// TIA Portal V20 export
TYPE "typeFDoorFunction"
// Safety status of door
// stored: Access Published, IsFailsafeCompliant true, Namespace Safety
   STRUCT
      fDoor1 { S7_SetPoint := 'True'} : "Safety.typeFDoorFunctionData";
      fDoor2 { S7_SetPoint := 'True'} : "Safety.typeFDoorFunctionData";   // Safety status of door
      fDoor3 { S7_SetPoint := 'True'} : "Safety.typeFDoorFunctionData";   // Safety status of door
      fDoor4 { S7_SetPoint := 'True'} : "Safety.typeFDoorFunctionData";   // Safety status of door
      fDoor5 { S7_SetPoint := 'True'} : "Safety.typeFDoorFunctionData";   // Safety status of door
      fDoor6 { S7_SetPoint := 'True'} : "Safety.typeFDoorFunctionData";   // Safety status of door
      fDoor7 { S7_SetPoint := 'True'} : "Safety.typeFDoorFunctionData";   // Safety status of door
      fDoor8 { S7_SetPoint := 'True'} : "Safety.typeFDoorFunctionData";   // Safety status of door
      fDoor9 { S7_SetPoint := 'True'} : "Safety.typeFDoorFunctionData";   // Safety status of door
   END_STRUCT;
END_TYPE
